TYPE
    ControlSignal1 :
    STRUCT
        word1 : word;
    END_STRUCT
END_TYPE

(* stored: Version 1.1.0.1, ProductVersion 3.1.4024.12
   DUT ControlSignal1: Id {40b6c50f-5807-440b-9ae8-21b6c9701ea5} *)
